FUNCTION_BLOCK FB_Light_tower_module
VAR_INPUT
END_VAR
VAR_OUTPUT
END_VAR
VAR
	lightTower	: ST_LightTower;

END_VAR

PROPERTY _lightTower : ST_LightTower
GET
_lightTower	:= lightTower;
END_GET
SET
lightTower	:= _lightTower;
END_SET
END_PROPERTY

{attribute 'TcRpcEnable'}
METHOD update_light_tower : BOOL
VAR_INPUT
	iLightTowerStatus	: UINT;
END_VAR
update_light_tower	:= FALSE;
lightTower.GREEN	:= iLightTowerStatus.0;
lightTower.RED		:= iLightTowerStatus.1;
lightTower.WHITE	:= iLightTowerStatus.2;
lightTower.BLUE		:= iLightTowerStatus.3;
lightTower.YELLOW	:= iLightTowerStatus.4;
lightTower.BUZZER	:= iLightTowerStatus.5;
update_light_tower	:= TRUE;
END_METHOD

END_FUNCTION_BLOCK

(* stored: Version 1.1.0.1, ProductVersion 3.1.4024.12
   POU FB_Light_tower_module: Id {76a2423a-0702-4258-b0ae-9c01d7e6ca39}, SpecialFunc None
   Property _lightTower: Id {f7d870eb-4a94-4b4b-89e4-8119c420cb86}
   Get Get: Id {7a0b5e46-296b-49e7-a384-a4950a54ec22}
   Set Set: Id {e6302abf-2dcb-4ed7-8096-c07360c2466b}
   Method update_light_tower: Id {972896c5-5b3b-459f-a81c-d8dd8173ee54} *)
